TEXTLIST TextList_VVAT_650_ETHERCAT
  0 = 'vanne' | FR: 'Vanne asservie' | EN: 'Servovalve'
  1 = 'max stab' | FR: 'Temps maximal de stabilisation' | EN: 'Maximum stabilization time'
  2 = 'alm stab' | FR: 'Surveillance pression - Temps avant alarme' | EN: 'Pressure supervision - Delay before alarm'
  3 = 'def stab' | FR: 'Surveillance pression - Temps avant défaut' | EN: 'Pressure supervision - Delay before fault'
  4 = 'pmin' | FR: 'Pression min. (mbar)' | EN: 'Min. pressure (mbar)'
  5 = 'pmax' | FR: 'Pression max. (mbar)' | EN: 'Max. pressure (mbar)'
  6 = 'TpsStab' | FR: 'Temps de stab.' | EN: 'Stab. time'
  7 = 'Pos' | FR: 'Position (%)' | EN: 'Position (%)'
  8 = 'Pression' | FR: 'Pression (mbar)' | EN: 'Pressure (mbar)'
   = ''
END_TEXTLIST

(* stored: Version 1.1.0.1, ProductVersion 3.1.4024.10
   TextList TextList_VVAT_650_ETHERCAT: Id {77163d7f-c3b9-4eff-84fc-335dfdc2aac1} *)
